# EPICS autosave request: dxp/branches/R3-0-branch/dxpApp/Db/dxp_settings.req
# FILE... dxp_settings.req
$(P)$(R)PeakingTime
#$(P)$(R)DynamicRange
$(P)$(R)TriggerThreshold
$(P)$(R)BaselineThreshold
$(P)$(R)BaselineCutPercent
$(P)$(R)BaselineCutEnable
$(P)$(R)BaselineFilterLength
$(P)$(R)EnergyThreshold
$(P)$(R)ADCPercentRule
$(P)$(R)MaxEnergy
$(P)$(R)PreampGain
$(P)$(R)DetectorPolarity
$(P)$(R)ResetDelay
$(P)$(R)GapTime
$(P)$(R)TriggerPeakingTime
$(P)$(R)TriggerGapTime
$(P)$(R)MaxWidth
$(P)$(R)ReadDXPParams.SCAN
$(P)$(R)TraceMode
$(P)$(R)TraceTime
$(P)$(R)BaselineHistogram.SCAN
$(P)$(R)TraceData.SCAN
$(P)SaveSystemFile
